{attribute 'GeneratedUsingTerminal: EJ7411-0000-0018'}
{attribute addProperty BoxType "EJ7411-0000-0018"}
{attribute addProperty Id "Following_error_actual_valueAT %I*DINT4"}
{attribute addProperty CRC "1520640191"}
{attribute addProperty Size "4"}
TYPE DRV_Following_error_actual_value_5AA320BF EXTENDS InputBase_8311D824 :
STRUCT
	{attribute addProperty Name "Following_error_actual_value"}
	Following_error_actual_value AT %I* : DINT;
END_STRUCT
END_TYPE

(* stored: Version 1.2.0.0, ProductVersion 3.1.4024.9
   DUT DRV_Following_error_actual_value_5AA320BF: Id {adbfa704-fdbf-413c-ae11-a072557cb616} *)
